(* CoDeSys 2.3 export: FTURNONK14PUMP.EXP *)

(* POU K14/fTurnOnK14Pump, ST *)
FUNCTION fTurnOnK14Pump : BOOL
VAR_INPUT
	PumpID : USINT;
END_VAR
VAR
END_VAR
	fSetK14Pump(TRUE, PumpID);
END_FUNCTION
